TYPE TYP_DEPRAG_AST11_HW_IN :
STRUCT
	Ready AT %I*: BOOL;
	OK AT %I*: BOOL;
	NOK AT %I*: BOOL;
END_STRUCT
END_TYPE

(* stored: Version 1.1.0.1, ProductVersion 3.1.4024.12
   DUT TYP_DEPRAG_AST11_HW_IN: Id {1d2d144e-acbc-4b4d-8a0d-747d857b1cf4} *)
